TYPE eTcoCarouselDirection :
(
	Cw := 0,
	Ccw := 1
);
END_TYPE

(* stored: Version 1.1.0.1
   DUT eTcoCarouselDirection: Id {9cbf3192-0a0c-0c90-3ed6-152529611f1c} *)
